(* CoDeSys 2.3 export: ATTR2_TU.EXP *)

(* Data type in Diag/Parameter *)
TYPE attr2_tu :
STRUCT
	MaxValue_s16		: INT;
(*
	InputChannel_u16	: UINT;
	ListEntries_u16	: UINT;
	data_au8 			: ARRAY [1..2] OF USINT;
*)
END_STRUCT
END_TYPE
